// TIA Portal project "Function Blocks" (V15.1)

(* hardware
DEVICE "S7-1200 station_1"  S7-1200 Station
   slot 0: "Rack_0"  S7-1200 Rack  Rack  V1.0
   slot 1: "S71214"  CPU 1214C DC/DC/DC  6ES7 214-1AG40-0XB0  V4.2
*)

// ===== PLC "S71214"  CPU 1214C DC/DC/DC =====

VAR_GLOBAL   // PLC tag table "Default tag table"
   "System_Byte" AT %MB1 : Byte;
   "FirstScan" AT %M1.0 : Bool;
   "DiagStatusUpdate" AT %M1.1 : Bool;
   "AlwaysTRUE" AT %M1.2 : Bool;
   "AlwaysFALSE" AT %M1.3 : Bool;
   "Clock_Byte" AT %MB0 : Byte;
   "Clock_10Hz" AT %M0.0 : Bool;
   "Clock_5Hz" AT %M0.1 : Bool;
   "Clock_2.5Hz" AT %M0.2 : Bool;
   "Clock_2Hz" AT %M0.3 : Bool;
   "Clock_1.25Hz" AT %M0.4 : Bool;
   "Clock_1Hz" AT %M0.5 : Bool;
   "Clock_0.625Hz" AT %M0.6 : Bool;
   "Clock_0.5Hz" AT %M0.7 : Bool;
   "M Count" AT %MW2 : Int;
   "M Start" AT %M4.0 : Bool;
   "T Trig 1" AT %M4.1 : Bool;
   "M Feedback 1" AT %M4.2 : Bool;
   "M Feedback 2" AT %M4.3 : Bool;
   "M Feedback 3" AT %M4.4 : Bool;
   "M Feedback 4" AT %M4.5 : Bool;
   "M Feedback 5" AT %M4.6 : Bool;
   "M Stop Restart" AT %M4.7 : Bool;
   "M Stop" AT %M5.0 : Bool;
   "M Stopped Feedback" AT %M5.1 : Bool;
   "M Start Backwash" AT %M5.2 : Bool;
   "T Trig 2" AT %M5.3 : Bool;
   "Filter Mode Active" AT %M5.4 : Bool;
   "M Filter Mode Active" AT %M5.5 : Bool;
   "Trig 1" AT %M5.6 : Bool;
   "M Valves Feedback" AT %M5.7 : Bool;
   "M Stage 1 Valves" AT %M6.0 : Bool;
   "M Start Feed Pump" AT %M6.1 : Bool;
   "M Forward Flush Done" AT %M6.2 : Bool;
   "M Open Next Valves" AT %M6.3 : Bool;
   "M Valve Feedback Stage 4" AT %M6.4 : Bool;
   "M Filtration Duration" AT %M6.5 : Bool;
   "M Startup Done" AT %M6.6 : Bool;
   "M Close Valves" AT %M6.7 : Bool;
   "M Valves Closed" AT %M7.0 : Bool;
   "M Open Backwash Valves 1" AT %M7.1 : Bool;
   "M Backwash Valve Feedback" AT %M7.2 : Bool;
   "M Open Air Release Valve" AT %M7.3 : Bool;
   "M Air Release Valve Open" AT %M7.4 : Bool;
   "M Start Blower" AT %M7.5 : Bool;
   "M Close Blower Valves" AT %M7.6 : Bool;
END_VAR

DATA_BLOCK "DB Sequence"   // DB1
{ S7_Optimized_Access := 'TRUE' }
VERSION : 0.1
   VAR
      "Stage Sequence" : Int;
      "Resume Sequence" : Int;
   END_VAR
BEGIN
END_DATA_BLOCK

DATA_BLOCK "FB_DOL_STARTER_DB"   // DB2
{ S7_Optimized_Access := 'TRUE' }
VERSION : 0.1
// stored: InstanceOfName FB_DOL_STARTER
"FB_DOL_STARTER"
BEGIN
END_DATA_BLOCK

DATA_BLOCK "Starter DB"   // DB3
{ S7_Optimized_Access := 'TRUE' }
VERSION : 0.1
   VAR
      "Emergency Stop Fault" : Bool;
      "Voltage Monitor Fault" : Bool;
      "Trip Fault" : Bool;
   END_VAR
   VAR RETAIN
      "Enable/Disable" : Bool;
      "Auto/Manual" : Bool;
   END_VAR
   VAR
      "Manual Start/Stop" : Bool;
   END_VAR
   VAR RETAIN
      "Auto Start" : Bool;
      "Manual Interlock" : Bool;
      "Auto Interlock" : Bool;
      "Duty Rotate Bit" : Bool;   // 1 if not used
      "Time Duration Controlled" : Bool;   // Yes = 1 , No = 0
      "On Duration" : Time;   // If Time Duration Control = 1
      "Off Duration" : Time;   // If Time Duration Control = 1
   END_VAR
   VAR
      "Q CMD" : Bool;
   END_VAR
   VAR RETAIN
      "Starter Status" : Word;
   END_VAR
BEGIN
END_DATA_BLOCK

FUNCTION_BLOCK "Stop Sequence"   // FB1, FBD
{ S7_Optimized_Access := 'TRUE' }
VERSION : 0.1
   VAR_INPUT
      "Stop Input with Restart" : Bool;
      "Stop Input Without Restart" : Bool;
      "Closed/Stopped Feedback" : Bool;
   END_VAR
   VAR_OUTPUT
      "Close/Stop Equipment" : Bool;
   END_VAR
   VAR_IN_OUT
      "Secuence Count" : Int;
   END_VAR
   VAR
      Restart : Bool;
      "Non Restart" : Bool;
      "Stop Done 1" : Bool;
      "Stop Done 2" : Bool;
   END_VAR
   VAR_TEMP   // added for the SCL form of the ladder/FBD networks
      _w1 : Bool;
      _w2 : Bool;
   END_VAR
BEGIN

REGION Network 1
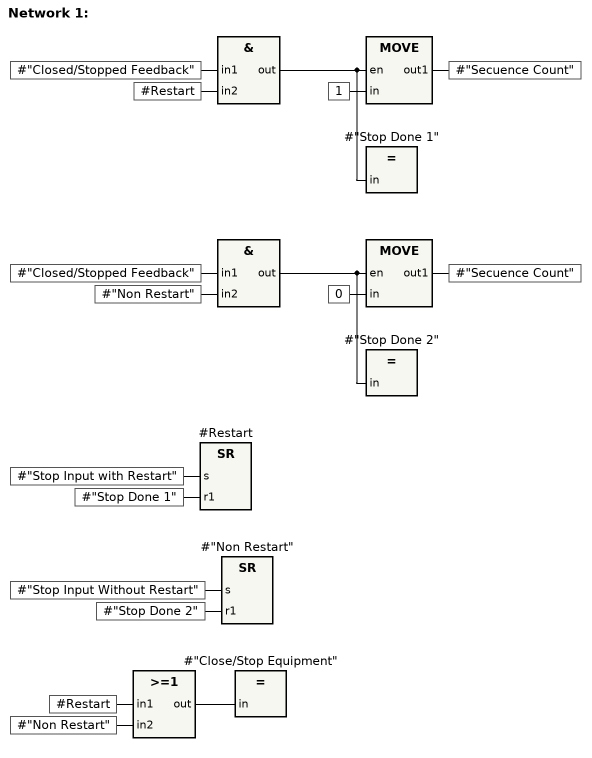
   #_w1 := #"Closed/Stopped Feedback" AND #Restart;
   IF #_w1 THEN #"Secuence Count" := 1; END_IF;
   #"Stop Done 1" := #_w1;
   #_w2 := #"Closed/Stopped Feedback" AND #"Non Restart";
   IF #_w2 THEN #"Secuence Count" := 0; END_IF;
   #"Stop Done 2" := #_w2;
   IF #"Stop Input with Restart" THEN
       #Restart := TRUE;   // SR flip-flop
   END_IF;
   IF #"Stop Done 1" THEN #Restart := FALSE; END_IF;
   IF #"Stop Input Without Restart" THEN
       #"Non Restart" := TRUE;   // SR flip-flop
   END_IF;
   IF #"Stop Done 2" THEN #"Non Restart" := FALSE; END_IF;
   #"Close/Stop Equipment" := #Restart OR #"Non Restart";
END_REGION
END_FUNCTION_BLOCK

FUNCTION_BLOCK "Stage"   // FB2, FBD
{ S7_Optimized_Access := 'TRUE' }
VERSION : 0.1
   VAR_INPUT
      "Stage Active" : Bool;
      "Time Delay Required" : Bool;
      "Stage Delay Time" : Time;
      "Feedback Required" : Bool;
      "Equipment Feedback" : Bool;
      "Delay Before Next Stage" : Bool;
      "Next Stage Delay" : Time;
      "Retain Output?" : Bool;
      "Reset Retain" : Bool;
   END_VAR
   VAR_OUTPUT
      "Stage Equipment Start" : Bool;
   END_VAR
   VAR_IN_OUT
      "Sequence Count" : Int;
   END_VAR
   VAR
      "Stage Timer" : TON_TIME;
      "Next Stage Timer" : TON_TIME;
      "Stage Equipment 1" : Bool;
      "Stage Equipment 2" : Bool;
      "Stage Euipment 3" : Bool;
      "Stage Equipment 4" : Bool;
   END_VAR
   VAR_TEMP   // added for the SCL form of the ladder/FBD networks
      _w1 : Bool;
   END_VAR
BEGIN

REGION Network 1
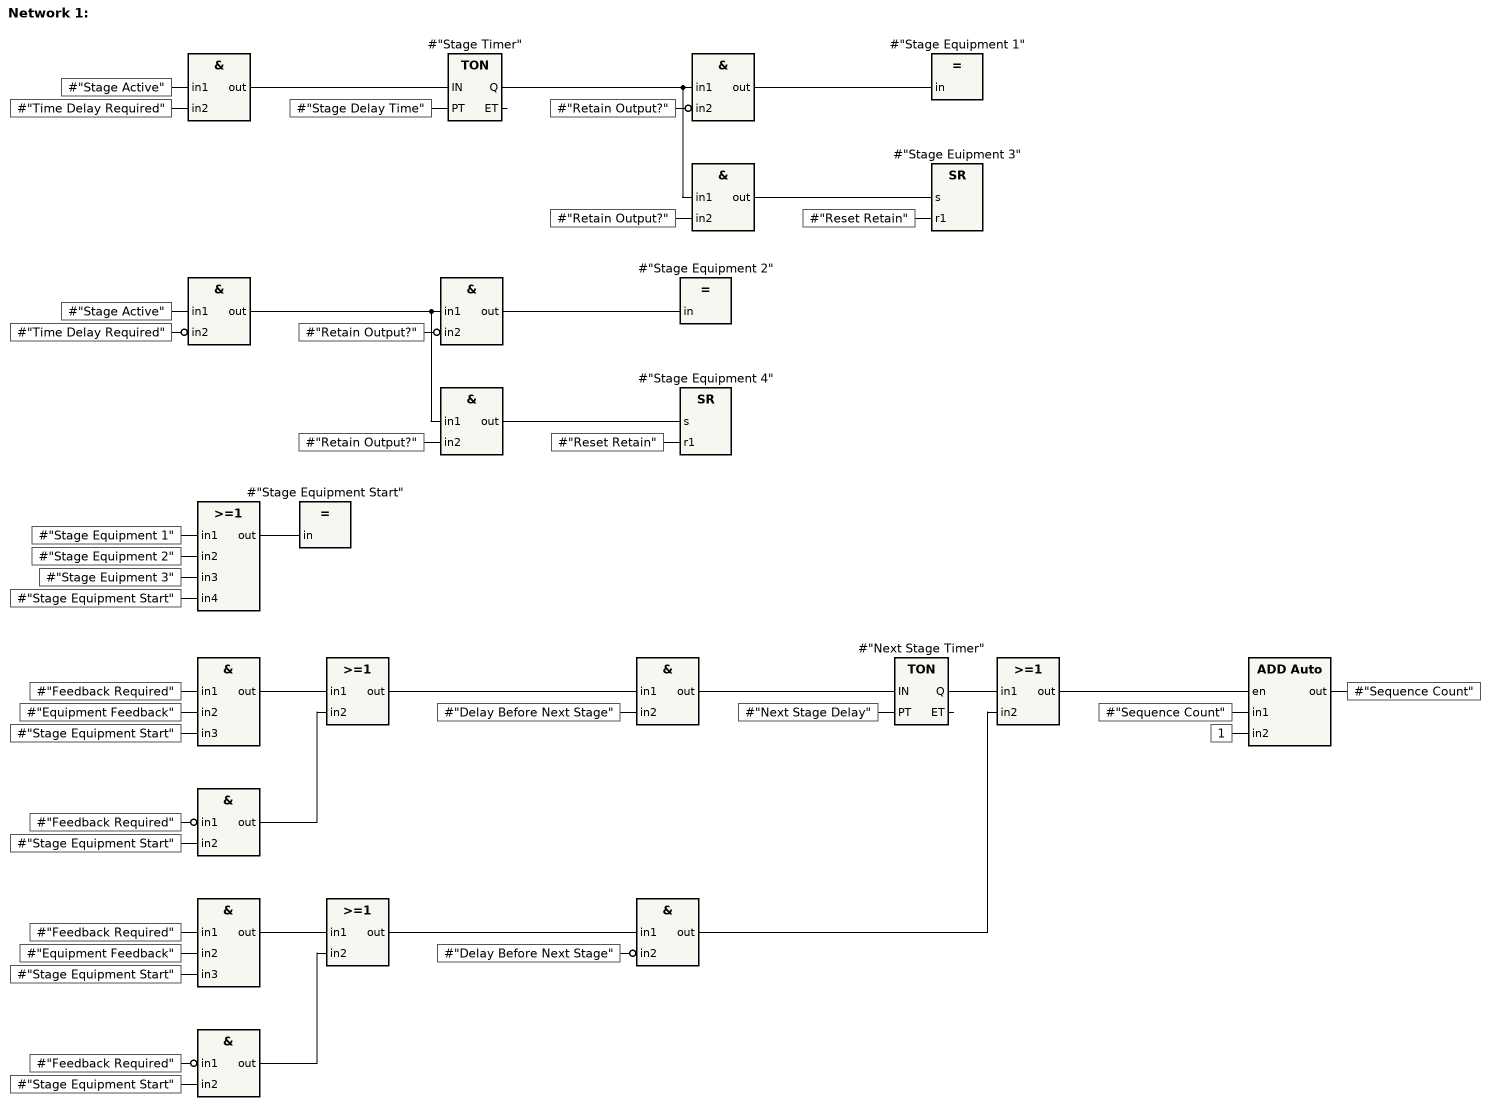
   #"Stage Timer"(IN := #"Stage Active" AND #"Time Delay Required", PT := #"Stage Delay Time");   // TON
   #"Stage Equipment 1" := #"Stage Timer".Q AND NOT #"Retain Output?";
   IF #"Stage Timer".Q AND #"Retain Output?" THEN
       #"Stage Euipment 3" := TRUE;   // SR flip-flop
   END_IF;
   IF #"Reset Retain" THEN #"Stage Euipment 3" := FALSE; END_IF;
   #_w1 := #"Stage Active" AND NOT #"Time Delay Required";
   #"Stage Equipment 2" := #_w1 AND NOT #"Retain Output?";
   IF #_w1 AND #"Retain Output?" THEN
       #"Stage Equipment 4" := TRUE;   // SR flip-flop
   END_IF;
   IF #"Reset Retain" THEN #"Stage Equipment 4" := FALSE; END_IF;
   #"Stage Equipment Start" := #"Stage Equipment 1" OR #"Stage Equipment 2" OR #"Stage Euipment 3" OR #"Stage Equipment Start";
   #"Next Stage Timer"(IN := ((#"Feedback Required" AND #"Equipment Feedback" AND #"Stage Equipment Start") OR (NOT #"Feedback Required" AND #"Stage Equipment Start")) AND #"Delay Before Next Stage",   // TON
                       PT := #"Next Stage Delay");
   IF #"Next Stage Timer".Q OR (((#"Feedback Required" AND #"Equipment Feedback" AND #"Stage Equipment Start") OR (NOT #"Feedback Required" AND #"Stage Equipment Start")) AND NOT #"Delay Before Next Stage") THEN
       #"Sequence Count" := #"Sequence Count" + 1;
   END_IF;
END_REGION
END_FUNCTION_BLOCK

FUNCTION_BLOCK "FB_DOL_STARTER"   // FB2, FBD
{ S7_Optimized_Access := 'TRUE' }
VERSION : 0.1
   VAR_INPUT
      EMERGENCY_STOP_FAULT : Bool;
      VOLTAGE_MONITOR_FAULT : Bool;
      MCB_AUX_FAULT : Bool;
      HMI_ENABLED_BOOL : Bool;
      HMI_AUTO_MAN_BOOL : Bool;   // AUTO = 1, MAN = 0
      HMI_MAN_START_BOOL : Bool;
      AUTO_START_BOOL : Bool;
      MAN_INTERLOCK_1 : Bool;
      MAN_INTERLOCK_2 : Bool;
      AUTO_INTERLOCK_1 : Bool;
      AUTO_INTERLOCK_2 : Bool;
      AUTO_INTERLOCK_3 : Bool;
      AUTO_INTERLOCK_4 : Bool;
      AUTO_INTERLOCK_5 : Bool;
      "DUTY_ROTATE_BIT (1 IF NOT USED)" : Bool;
      "TIME_DUR_CONTROLLED (YES=1,NO=0)" : Bool;
      ON_DURATION : Time;
      OFF_DURATION : Time;
   END_VAR
   VAR_OUTPUT
      STARTER_STATUS : Word;
   END_VAR
   VAR_IN_OUT
      Q_CMD : Bool;
   END_VAR
   VAR
      "HEALTH STATUS" : Bool;
      "MANUAL EN" : Bool;
      "AUTO EN" : Bool;
      MAN_TRIG_1 : Bool;
      MAN_TRIG_2 : Bool;
      IEC_Timer_0_Instance : TON_TIME;
      IEC_Timer_0_Instance_1 : TON_TIME;
      AUTO_TRIG_1 : Bool;
      AUTO_TRIG_2 : Bool;
   END_VAR
   VAR_TEMP   // added for the SCL form of the ladder/FBD networks
      _w1 : Bool;
      _w2 : Bool;
      _w3 : Bool;
   END_VAR
BEGIN

REGION Network 1: Healthy Starter
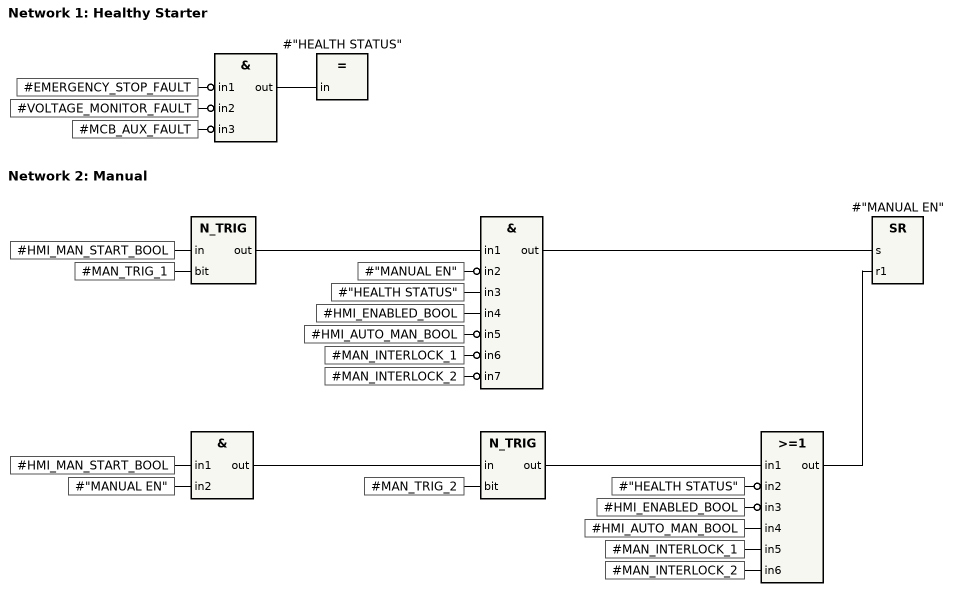
   #"HEALTH STATUS" := NOT #EMERGENCY_STOP_FAULT AND NOT #VOLTAGE_MONITOR_FAULT AND NOT #MCB_AUX_FAULT;
END_REGION

REGION Network 2: Manual
   #_w1 := NOT #HMI_MAN_START_BOOL AND #MAN_TRIG_1;   // falling edge
   #MAN_TRIG_1 := #HMI_MAN_START_BOOL;
   #_w2 := #HMI_MAN_START_BOOL AND #"MANUAL EN";
   #_w3 := NOT #_w2 AND #MAN_TRIG_2;   // falling edge
   #MAN_TRIG_2 := #_w2;
   IF #_w1 AND NOT #"MANUAL EN" AND #"HEALTH STATUS" AND #HMI_ENABLED_BOOL AND NOT #HMI_AUTO_MAN_BOOL AND NOT #MAN_INTERLOCK_1 AND NOT #MAN_INTERLOCK_2 THEN
       #"MANUAL EN" := TRUE;   // SR flip-flop
   END_IF;
   IF #_w3 OR NOT #"HEALTH STATUS" OR NOT #HMI_ENABLED_BOOL OR #HMI_AUTO_MAN_BOOL OR #MAN_INTERLOCK_1 OR #MAN_INTERLOCK_2 THEN
       #"MANUAL EN" := FALSE;
   END_IF;
END_REGION

REGION Network 3: Auto
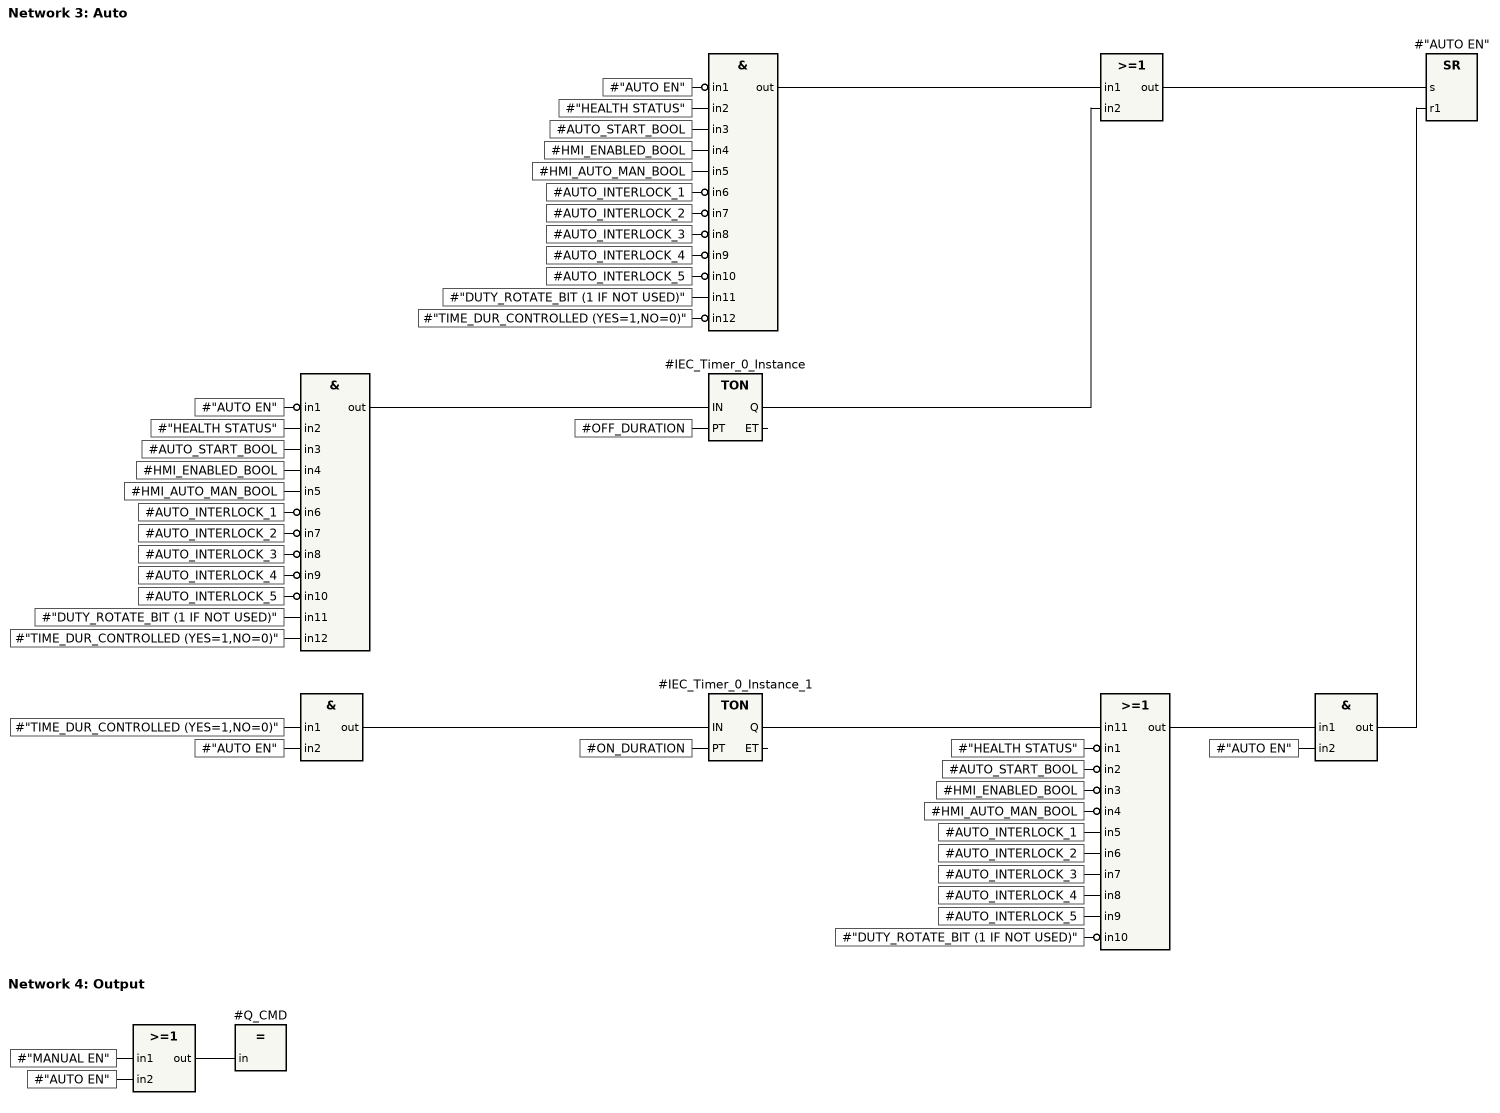
   #IEC_Timer_0_Instance(IN := NOT #"AUTO EN" AND #"HEALTH STATUS" AND #AUTO_START_BOOL AND #HMI_ENABLED_BOOL AND #HMI_AUTO_MAN_BOOL AND NOT #AUTO_INTERLOCK_1 AND NOT #AUTO_INTERLOCK_2 AND NOT #AUTO_INTERLOCK_3 AND NOT #AUTO_INTERLOCK_4 AND NOT #AUTO_INTERLOCK_5 AND #"DUTY_ROTATE_BIT (1 IF NOT USED)" AND #"TIME_DUR_CONTROLLED (YES=1,NO=0)",   // TON
                         PT := #OFF_DURATION);
   #IEC_Timer_0_Instance_1(IN := #"TIME_DUR_CONTROLLED (YES=1,NO=0)" AND #"AUTO EN", PT := #ON_DURATION);   // TON
   #_w1 := (#IEC_Timer_0_Instance_1.Q OR NOT #"HEALTH STATUS" OR NOT #AUTO_START_BOOL OR NOT #HMI_ENABLED_BOOL OR NOT #HMI_AUTO_MAN_BOOL OR #AUTO_INTERLOCK_1 OR #AUTO_INTERLOCK_2 OR #AUTO_INTERLOCK_3 OR #AUTO_INTERLOCK_4 OR #AUTO_INTERLOCK_5 OR NOT #"DUTY_ROTATE_BIT (1 IF NOT USED)") AND #"AUTO EN";
   IF (NOT #"AUTO EN" AND #"HEALTH STATUS" AND #AUTO_START_BOOL AND #HMI_ENABLED_BOOL AND #HMI_AUTO_MAN_BOOL AND NOT #AUTO_INTERLOCK_1 AND NOT #AUTO_INTERLOCK_2 AND NOT #AUTO_INTERLOCK_3 AND NOT #AUTO_INTERLOCK_4 AND NOT #AUTO_INTERLOCK_5 AND #"DUTY_ROTATE_BIT (1 IF NOT USED)" AND NOT #"TIME_DUR_CONTROLLED (YES=1,NO=0)") OR #IEC_Timer_0_Instance.Q THEN
       #"AUTO EN" := TRUE;   // SR flip-flop
   END_IF;
   IF #_w1 THEN #"AUTO EN" := FALSE; END_IF;
END_REGION

REGION Network 4: Output
   #Q_CMD := #"MANUAL EN" OR #"AUTO EN";
END_REGION

REGION Network 5: Status
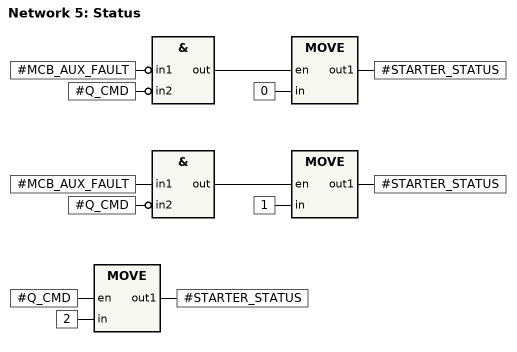
   IF NOT #MCB_AUX_FAULT AND NOT #Q_CMD THEN #STARTER_STATUS := 0; END_IF;
   IF #MCB_AUX_FAULT AND NOT #Q_CMD THEN #STARTER_STATUS := 1; END_IF;
   IF #Q_CMD THEN #STARTER_STATUS := 2; END_IF;
END_REGION
END_FUNCTION_BLOCK

FUNCTION_BLOCK "Last Stage"   // FB3, FBD
{ S7_Optimized_Access := 'TRUE' }
VERSION : 0.1
   VAR_INPUT
      "Stage Active" : Bool;
      "Time Delay Required" : Bool;
      "Stage Delay Time" : Time;
      "Feedback Required" : Bool;
      "Equipment Feedback" : Bool;
      "Delay Before Next Stage" : Bool;
   END_VAR
   VAR_OUTPUT
      "Stage Equipment Start" : Bool;
   END_VAR
   VAR_IN_OUT
      "Sequence Count" : Int;
   END_VAR
   VAR
      "Stage Timer" : TON_TIME;
      "Stage Equipment 1" : Bool;
      "Stage Equipment 2" : Bool;
   END_VAR
BEGIN

REGION Network 1
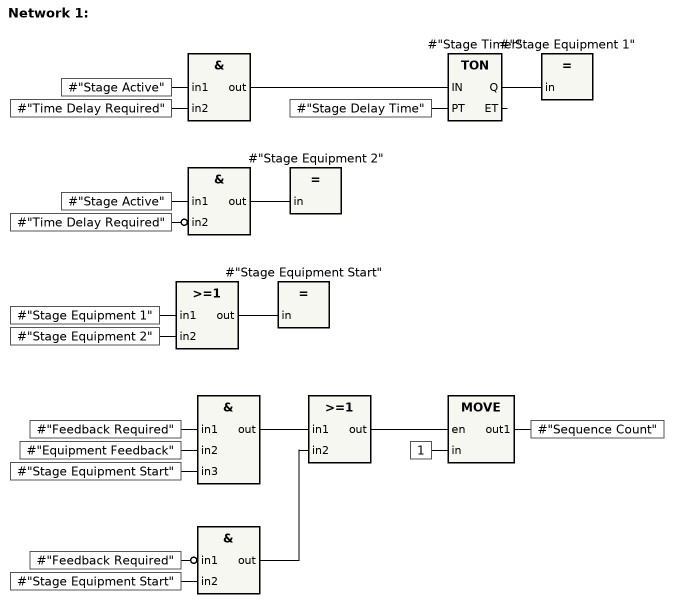
   #"Stage Timer"(IN := #"Stage Active" AND #"Time Delay Required", PT := #"Stage Delay Time");   // TON
   #"Stage Equipment 1" := #"Stage Timer".Q;
   #"Stage Equipment 2" := #"Stage Active" AND NOT #"Time Delay Required";
   #"Stage Equipment Start" := #"Stage Equipment 1" OR #"Stage Equipment 2";
   IF (#"Feedback Required" AND #"Equipment Feedback" AND #"Stage Equipment Start") OR (NOT #"Feedback Required" AND #"Stage Equipment Start") THEN
       #"Sequence Count" := 1;
   END_IF;
END_REGION
END_FUNCTION_BLOCK

FUNCTION "FC DOL Starter" : Void   // FC2, FBD
{ S7_Optimized_Access := 'TRUE' }
VERSION : 0.1
BEGIN

REGION Network 1: Starter
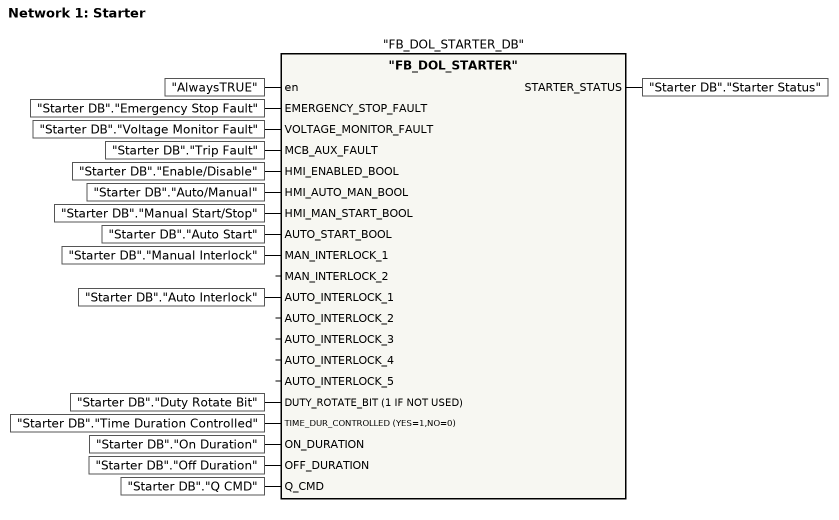
   IF "AlwaysTRUE" THEN
       "FB_DOL_STARTER_DB"(EMERGENCY_STOP_FAULT := "Starter DB"."Emergency Stop Fault",   // "FB_DOL_STARTER"
                           VOLTAGE_MONITOR_FAULT := "Starter DB"."Voltage Monitor Fault",
                           MCB_AUX_FAULT := "Starter DB"."Trip Fault",
                           HMI_ENABLED_BOOL := "Starter DB"."Enable/Disable",
                           HMI_AUTO_MAN_BOOL := "Starter DB"."Auto/Manual",
                           HMI_MAN_START_BOOL := "Starter DB"."Manual Start/Stop",
                           AUTO_START_BOOL := "Starter DB"."Auto Start",
                           MAN_INTERLOCK_1 := "Starter DB"."Manual Interlock",
                           AUTO_INTERLOCK_1 := "Starter DB"."Auto Interlock",
                           "DUTY_ROTATE_BIT (1 IF NOT USED)" := "Starter DB"."Duty Rotate Bit",
                           "TIME_DUR_CONTROLLED (YES=1,NO=0)" := "Starter DB"."Time Duration Controlled",
                           ON_DURATION := "Starter DB"."On Duration",
                           OFF_DURATION := "Starter DB"."Off Duration",
                           Q_CMD := "Starter DB"."Q CMD",
                           STARTER_STATUS => "Starter DB"."Starter Status");
   END_IF;
END_REGION
END_FUNCTION

ORGANIZATION_BLOCK "Main"   // OB1, LAD, ProgramCycle
TITLE = "Main Program Sweep (Cycle)"
{ S7_Optimized_Access := 'TRUE' }
VERSION : 0.1
   VAR_INPUT
      Initial_Call : Bool;   // Initial call of this OB
      Remanence : Bool;   // =True, if remanent data are available
   END_VAR
   VAR_TEMP
      "Feedback 1" : Bool;
      "Feedback 2" : Bool;
      "Feedback 3" : Bool;
      "Feedback 4" : Bool;
      "Feedback 5" : Bool;
   END_VAR
BEGIN
END_ORGANIZATION_BLOCK

// folder: Herbertsdale

FUNCTION "FC Herbertsdale Sequence" : Void   // FC1, FBD
{ S7_Optimized_Access := 'TRUE' }
VERSION : 0.1
BEGIN
END_FUNCTION